(* Schneider Machine Expert - Basic project Seren_Alarm, file version 3.0.0.0 *)

HARDWARE
  Cpu 0: TM221CE16R
  EthernetConfiguration: NetworkName=M221, IpAllocationMode=FixedAddress, IpAddress=192.168.0.221, SubnetMask=255.255.255.0
  SerialLineConfiguration: Baud=Baud19200, Parity=ParityEven, DataBits=DataBits8, StopBits=StopBits1, PhysicalMedium=PhysicalMediumRs485, TransmissionMode=TransmissionModeModbusRtu, SlaveId=1, Addressing=SlaveAddressing
  MastTask: UsePeriodScanMode=true, PeriodScan=10
  FastTask: Period=255
  CpuBehavior: StartingMode=StartInRun, AutoSaveRamOnEeprom=true, WatchdogPeriod=250

SYMBOLS  (address, symbol, comment, settings)
  %M0       M_COM_OK
  %M1       M_HB_LAST
  %M2       M_HB_TOGGLED
  %M10      M_ENABLE_GEN
  %M11      M_PULSE_OUT
  %M12      M_PAUSE_OUT
  %M13      M_SERIES_PAUSE
  %S12      SB_RUNMODE  "The controller is running"
  %MW0      PLC_CONTROL_WORD
  %MW1      PLC_STATUS_WORD
  %MW2      SOUND_PROFILE_CODE
  %MW3      SOUND_PULSE_COUNT
  %MW4      SOUND_PULSE_TIME_MS
  %MW5      SOUND_PAUSE_TIME_MS
  %MW6      SOUND_SERIES_INTERVAL_MS
  %MW10     ACTIVE_PULSE_COUNT
  %MW11     ACTIVE_PULSE_T_PRESET
  %MW12     ACTIVE_PAUSE_T_PRESET
  %MW13     ACTIVE_SERIES_T_PRESET
  %MW14     SERIES_COUNTER_VAL
  %TM0        [Preset=12, Base=OneSecond]
  %TM1        [Preset=20, Base=TenMilliSeconds]
  %TM2        [Preset=30, Base=TenMilliSeconds]
  %TM3        [Preset=5, Base=OneSecond]
  %QWM0     QW_HEARD_BEAT_WORD
  %QWM1     QW_PLC_CONTROL_WORD
  %IWM0     IW_PLC_HEARD_BEAT_WORD
  %IWM1     IW_PLC_STATUS_WORD

POU SIREN_CONTROL
  (* SectionNumber=1 *)

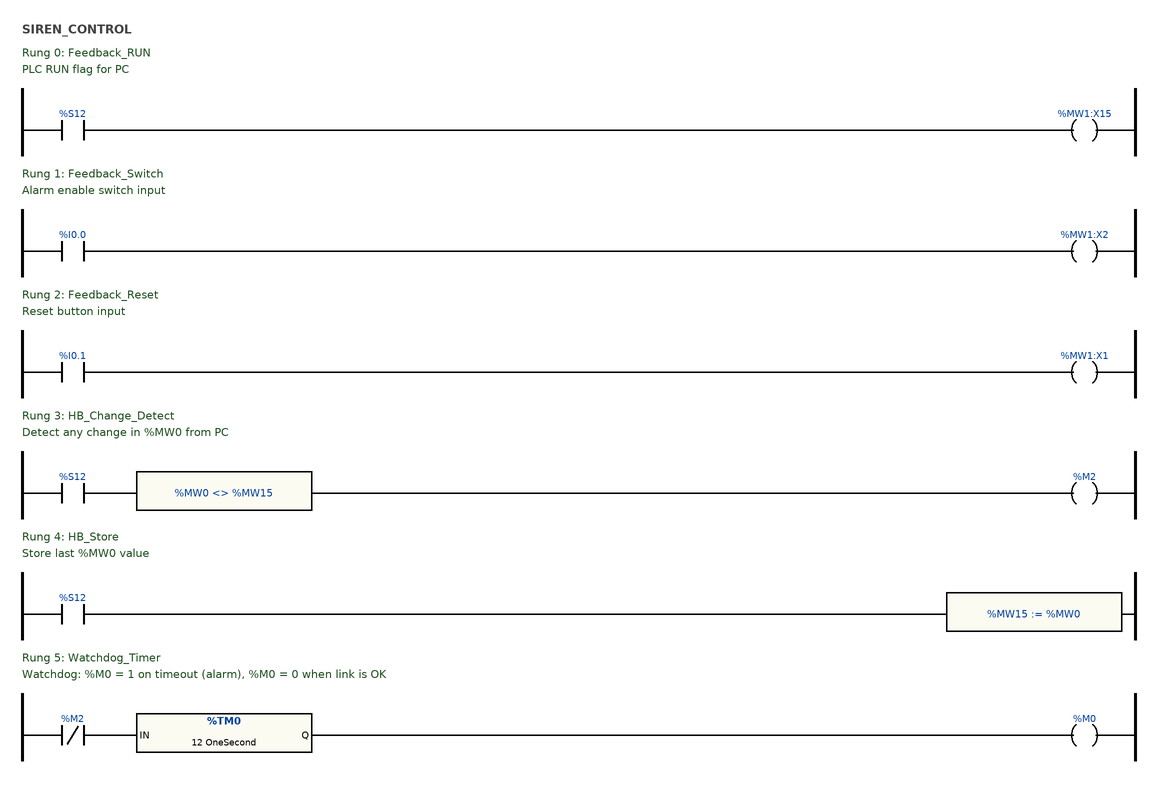

// Rung 0: Feedback_RUN
// PLC RUN flag for PC
  LD %S12                 (* SB_RUNMODE *)
  ST %MW1:X15             (* PLC_STATUS_WORD *)
  // as ST:
  //   PLC_STATUS_WORD:X15 := SB_RUNMODE;

// Rung 1: Feedback_Switch
// Alarm enable switch input
  LD %I0.0
  ST %MW1:X2              (* PLC_STATUS_WORD *)
  // as ST:
  //   PLC_STATUS_WORD:X2 := %I0.0;

// Rung 2: Feedback_Reset
// Reset button input
  LD %I0.1
  ST %MW1:X1              (* PLC_STATUS_WORD *)
  // as ST:
  //   PLC_STATUS_WORD:X1 := %I0.1;

// Rung 3: HB_Change_Detect
// Detect any change in %MW0 from PC
  LD %S12                 (* SB_RUNMODE *)
  AND [ %MW0 <> %MW15 ]   (* PLC_CONTROL_WORD *)
  ST %M2                  (* M_HB_TOGGLED *)
  // as ST:
  //   M_HB_TOGGLED := SB_RUNMODE AND PLC_CONTROL_WORD <> %MW15;

// Rung 4: HB_Store
// Store last %MW0 value
  LD %S12                 (* SB_RUNMODE *)
  [ %MW15 := %MW0 ]       (* PLC_CONTROL_WORD *)
  // as ST:
  //   IF SB_RUNMODE THEN %MW15 := PLC_CONTROL_WORD; END_IF;

// Rung 5: Watchdog_Timer
// Watchdog: %M0 = 1 on timeout (alarm), %M0 = 0 when link is OK
  BLK %TM0
  LDN %M2                 (* M_HB_TOGGLED *)
  IN
  OUT_BLK
  LD Q
  ST %M0                  (* M_COM_OK *)
  END_BLK
  // as ST:
  //   %TM0(IN := NOT M_HB_TOGGLED);
  //   M_COM_OK := %TM0.Q;

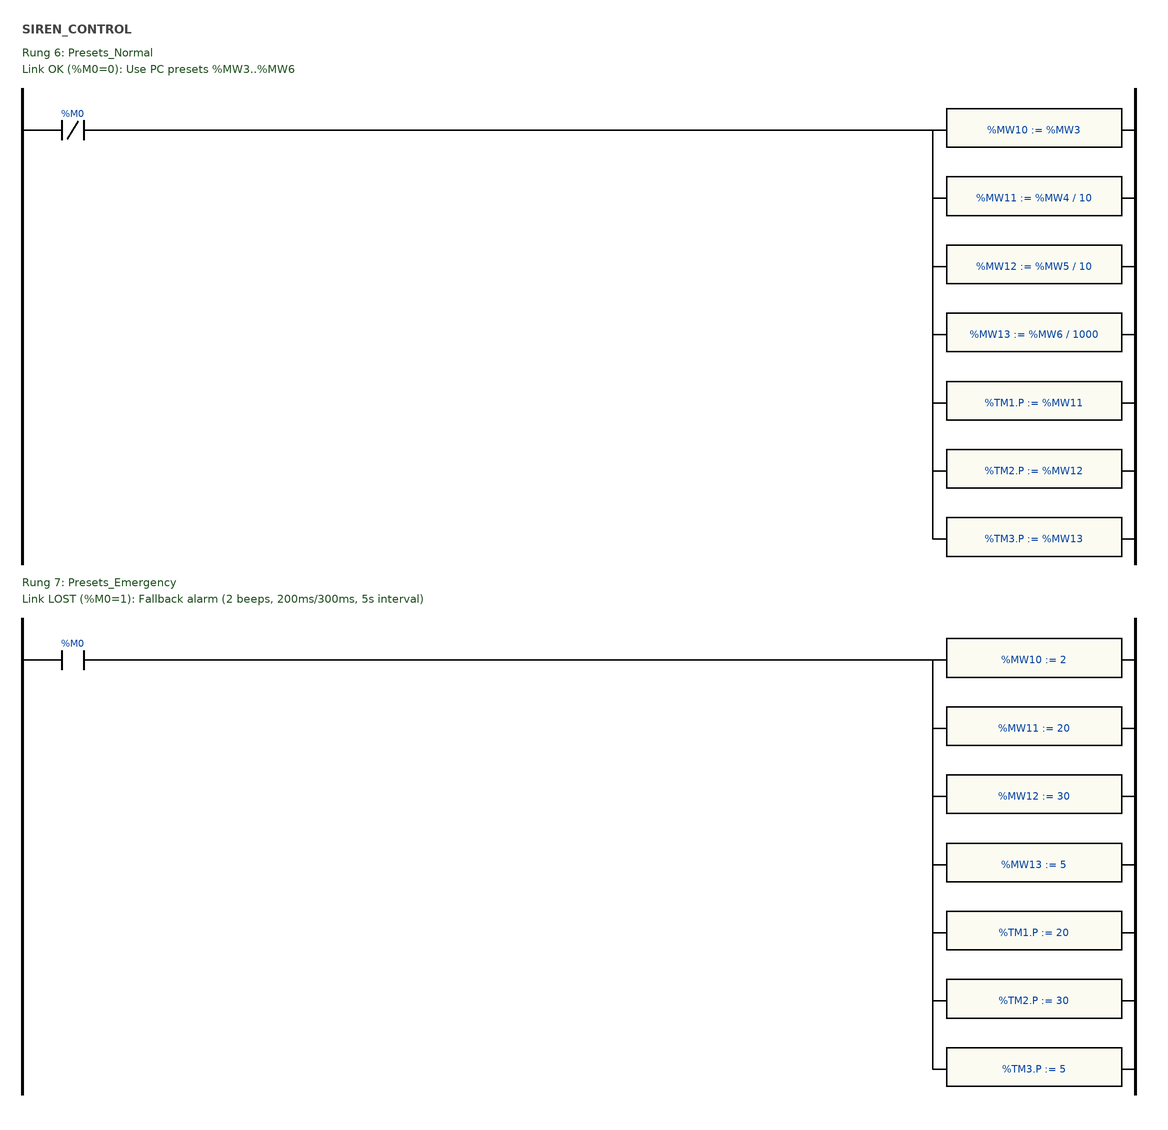

// Rung 6: Presets_Normal
// Link OK (%M0=0): Use PC presets %MW3..%MW6
  LDN %M0                 (* M_COM_OK *)
  [ %MW10 := %MW3 ]       (* ACTIVE_PULSE_COUNT, SOUND_PULSE_COUNT *)
  [ %MW11 := %MW4 / 10 ]  (* ACTIVE_PULSE_T_PRESET, SOUND_PULSE_TIME_MS *)
  [ %MW12 := %MW5 / 10 ]  (* ACTIVE_PAUSE_T_PRESET, SOUND_PAUSE_TIME_MS *)
  [ %MW13 := %MW6 / 1000 ](* ACTIVE_SERIES_T_PRESET, SOUND_SERIES_INTERVAL_MS *)
  [ %TM1.P := %MW11 ]     (* ACTIVE_PULSE_T_PRESET *)
  [ %TM2.P := %MW12 ]     (* ACTIVE_PAUSE_T_PRESET *)
  [ %TM3.P := %MW13 ]     (* ACTIVE_SERIES_T_PRESET *)
  // as ST:
  //   IF NOT M_COM_OK THEN ACTIVE_PULSE_COUNT := SOUND_PULSE_COUNT; END_IF;
  //   IF NOT M_COM_OK THEN ACTIVE_PULSE_T_PRESET := SOUND_PULSE_TIME_MS / 10; END_IF;
  //   IF NOT M_COM_OK THEN ACTIVE_PAUSE_T_PRESET := SOUND_PAUSE_TIME_MS / 10; END_IF;
  //   IF NOT M_COM_OK THEN ACTIVE_SERIES_T_PRESET := SOUND_SERIES_INTERVAL_MS / 1000; END_IF;
  //   IF NOT M_COM_OK THEN %TM1.P := ACTIVE_PULSE_T_PRESET; END_IF;
  //   IF NOT M_COM_OK THEN %TM2.P := ACTIVE_PAUSE_T_PRESET; END_IF;
  //   IF NOT M_COM_OK THEN %TM3.P := ACTIVE_SERIES_T_PRESET; END_IF;

// Rung 7: Presets_Emergency
// Link LOST (%M0=1): Fallback alarm (2 beeps, 200ms/300ms, 5s interval)
  LD %M0                  (* M_COM_OK *)
  [ %MW10 := 2 ]          (* ACTIVE_PULSE_COUNT *)
  [ %MW11 := 20 ]         (* ACTIVE_PULSE_T_PRESET *)
  [ %MW12 := 30 ]         (* ACTIVE_PAUSE_T_PRESET *)
  [ %MW13 := 5 ]          (* ACTIVE_SERIES_T_PRESET *)
  [ %TM1.P := 20 ]
  [ %TM2.P := 30 ]
  [ %TM3.P := 5 ]
  // as ST:
  //   IF M_COM_OK THEN ACTIVE_PULSE_COUNT := 2; END_IF;
  //   IF M_COM_OK THEN ACTIVE_PULSE_T_PRESET := 20; END_IF;
  //   IF M_COM_OK THEN ACTIVE_PAUSE_T_PRESET := 30; END_IF;
  //   IF M_COM_OK THEN ACTIVE_SERIES_T_PRESET := 5; END_IF;
  //   IF M_COM_OK THEN %TM1.P := 20; END_IF;
  //   IF M_COM_OK THEN %TM2.P := 30; END_IF;
  //   IF M_COM_OK THEN %TM3.P := 5; END_IF;

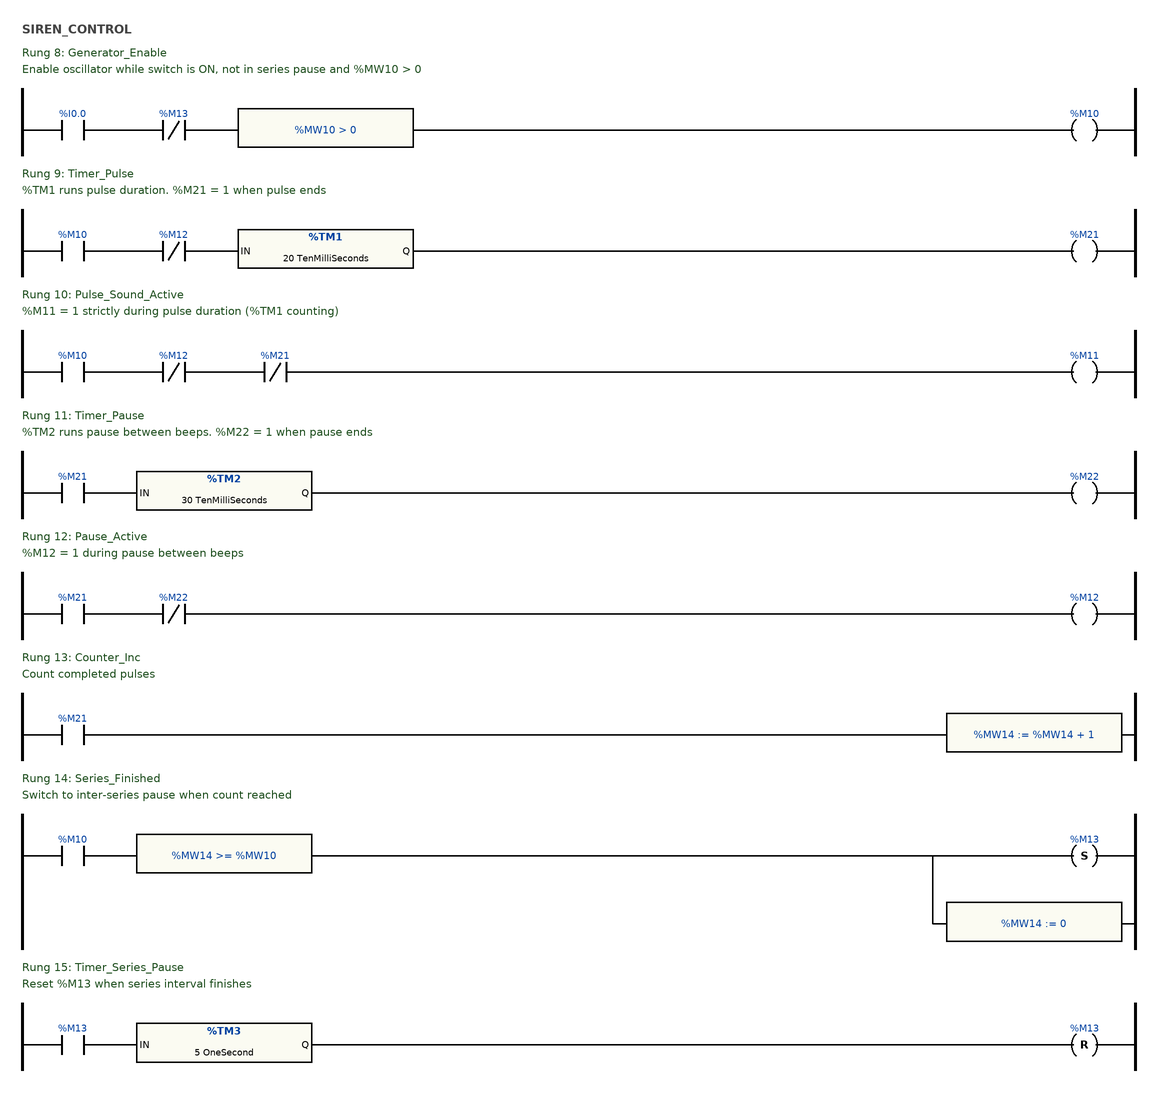

// Rung 8: Generator_Enable
// Enable oscillator while switch is ON, not in series pause and %MW10 > 0
  LD %I0.0
  ANDN %M13               (* M_SERIES_PAUSE *)
  AND [ %MW10 > 0 ]       (* ACTIVE_PULSE_COUNT *)
  ST %M10                 (* M_ENABLE_GEN *)
  // as ST:
  //   M_ENABLE_GEN := %I0.0 AND NOT M_SERIES_PAUSE AND ACTIVE_PULSE_COUNT > 0;

// Rung 9: Timer_Pulse
// %TM1 runs pulse duration. %M21 = 1 when pulse ends
  BLK %TM1
  LD %M10                 (* M_ENABLE_GEN *)
  ANDN %M12               (* M_PAUSE_OUT *)
  IN
  OUT_BLK
  LD Q
  ST %M21
  END_BLK
  // as ST:
  //   %TM1(IN := M_ENABLE_GEN AND NOT M_PAUSE_OUT);
  //   %M21 := %TM1.Q;

// Rung 10: Pulse_Sound_Active
// %M11 = 1 strictly during pulse duration (%TM1 counting)
  LD %M10                 (* M_ENABLE_GEN *)
  ANDN %M12               (* M_PAUSE_OUT *)
  ANDN %M21
  ST %M11                 (* M_PULSE_OUT *)
  // as ST:
  //   M_PULSE_OUT := M_ENABLE_GEN AND NOT M_PAUSE_OUT AND NOT %M21;

// Rung 11: Timer_Pause
// %TM2 runs pause between beeps. %M22 = 1 when pause ends
  BLK %TM2
  LD %M21
  IN
  OUT_BLK
  LD Q
  ST %M22
  END_BLK
  // as ST:
  //   %TM2(IN := %M21);
  //   %M22 := %TM2.Q;

// Rung 12: Pause_Active
// %M12 = 1 during pause between beeps
  LD %M21
  ANDN %M22
  ST %M12                 (* M_PAUSE_OUT *)
  // as ST:
  //   M_PAUSE_OUT := %M21 AND NOT %M22;

// Rung 13: Counter_Inc
// Count completed pulses
  LD %M21
  [ %MW14 := %MW14 + 1 ]  (* SERIES_COUNTER_VAL, SERIES_COUNTER_VAL *)
  // as ST:
  //   IF %M21 THEN SERIES_COUNTER_VAL := SERIES_COUNTER_VAL + 1; END_IF;

// Rung 14: Series_Finished
// Switch to inter-series pause when count reached
  LD %M10                 (* M_ENABLE_GEN *)
  AND [ %MW14 >= %MW10 ]  (* SERIES_COUNTER_VAL, ACTIVE_PULSE_COUNT *)
  S %M13                  (* M_SERIES_PAUSE *)
  [ %MW14 := 0 ]          (* SERIES_COUNTER_VAL *)
  // as ST:
  //   IF M_ENABLE_GEN AND SERIES_COUNTER_VAL >= ACTIVE_PULSE_COUNT THEN M_SERIES_PAUSE := TRUE; END_IF;
  //   IF M_ENABLE_GEN AND SERIES_COUNTER_VAL >= ACTIVE_PULSE_COUNT THEN SERIES_COUNTER_VAL := 0; END_IF;

// Rung 15: Timer_Series_Pause
// Reset %M13 when series interval finishes
  BLK %TM3
  LD %M13                 (* M_SERIES_PAUSE *)
  IN
  OUT_BLK
  LD Q
  R %M13                  (* M_SERIES_PAUSE *)
  END_BLK
  // as ST:
  //   %TM3(IN := M_SERIES_PAUSE);
  //   IF %TM3.Q THEN M_SERIES_PAUSE := FALSE; END_IF;

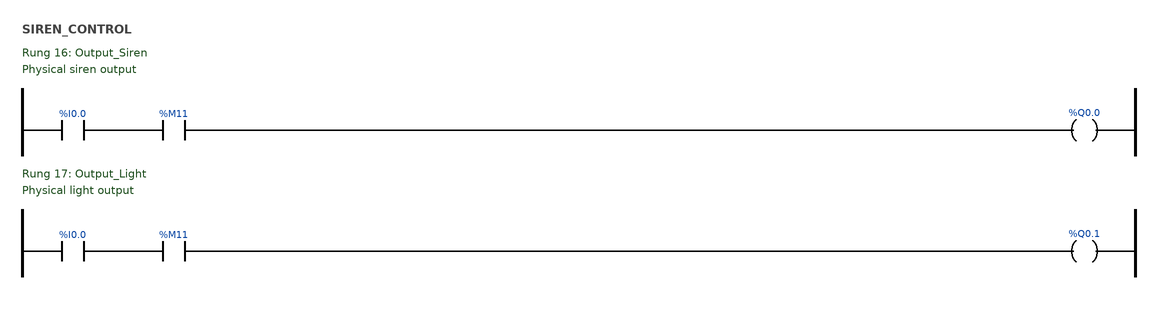

// Rung 16: Output_Siren
// Physical siren output
  LD %I0.0
  AND %M11                (* M_PULSE_OUT *)
  ST %Q0.0
  // as ST:
  //   %Q0.0 := %I0.0 AND M_PULSE_OUT;

// Rung 17: Output_Light
// Physical light output
  LD %I0.0
  AND %M11                (* M_PULSE_OUT *)
  ST %Q0.1
  // as ST:
  //   %Q0.1 := %I0.0 AND M_PULSE_OUT;
